{attribute addProperty BoxType "EK1122-0000-0018"}
{attribute addProperty Id "Beckhoff_EL1xxxsub_EK1100EK1100_179A0949162"}
{attribute addProperty CRC "3124704701"}
{attribute addProperty SizeInBites "16"}
{attribute addProperty SizeInBytes "2"}
TYPE Beckhoff_EL1xxxEK1122_BA3F35BD EXTENDS EK1122_179A0949 :
STRUCT
	{attribute addProperty Name "Beckhoff_EL1xxxsub_EK1100"}
	Beckhoff_EL1xxxsub_EK1100 : EK1100_179A0949;
END_STRUCT
END_TYPE

(* stored: Version 1.2.0.0, ProductVersion 3.1.4024.9
   DUT Beckhoff_EL1xxxEK1122_BA3F35BD: Id {d102f5d6-c5bb-46b8-839a-4e83d6b9989f} *)
